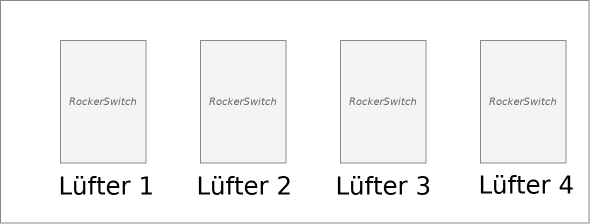
VISUALIZATION Visualisierung  // 590x224
    Label (45,150 123x72), "Lüfter 1"
    RockerSwitch (60,40 86x123), variable: VISU.Luefter_1, behaviour: TOGGLE, style: Switch-RockerSwitch-Gray
    Label (183,150 123x72), "Lüfter 2"
    RockerSwitch (200,40 86x123), variable: VISU.Luefter_2, behaviour: TOGGLE, style: Switch-RockerSwitch-Gray
    Label (322,150 123x72), "Lüfter 3"
    RockerSwitch (340,40 86x123), variable: VISU.Luefter_3, behaviour: TOGGLE, style: Switch-RockerSwitch-Gray
    Label (465,149 123x72), "Lüfter 4"
    RockerSwitch (480,40 86x123), variable: VISU.Luefter_4, behaviour: TOGGLE, style: Switch-RockerSwitch-Gray
END_VISUALIZATION

(* stored: Version 1.1.0.1, ProductVersion 3.1.4022.6
   Visu Visualisierung: Id {258ce351-fc62-45d1-9ff7-a94ff2a9643e} *)
